TEXTLIST TL_TerminalType
  0 = 'NoTerminal'
  1001 = 'KL300x'
  1002 = 'KL301x'
  1003 = 'KL302x'
  1004 = 'KL304x'
  1005 = 'KL305x'
  1006 = 'KL306x'
  1007 = 'KL310x'
  1008 = 'KL311x'
  1009 = 'KL312x'
  1010 = 'KL313x'
  1011 = 'KL314x'
  1012 = 'KL315x'
  1013 = 'KL317x'
  1014 = 'KL318x'
  1015 = 'KL340x'
  1016 = 'KL344x'
  1017 = 'KL346x'
  1018 = 'KL331x'
  2001 = 'EL331x'
  2002 = 'EL320x'
  2003 = 'EL316x'
  3001 = 'FM33xx'
  3002 = 'EM8908'
  10000 = 'Customized'
   = ''
END_TEXTLIST

(* stored: Version 1.1.0.1, ProductVersion 3.1.4020.12
   TextList TL_TerminalType: Id {0b12124f-5541-4cb9-a99e-d67611517983} *)
